# EPICS autosave request: CAENV895/iocBoot/iocCAENV895-IOC-01/vmeconfigMenu.req
file configMenu.req P=$(P),CONFIG=$(CONFIG)
file vmeconfig_settings.req
